// TIA Portal V19 export
TYPE "LubrValve_HMI"
// stored: Access Published
   STRUCT
      ManReq : Bool;
      AutoReq : Bool;
      Running : Bool;
      Alarm : Bool;
      ActualWorkTime : Time;
   END_STRUCT;
END_TYPE
